PROGRAM P_Sortierer
VAR
END_VAR

(* 
Baustein: FC24 Sortierer
Zeitstempel Code: 25.06.2018 11:16:45
Interface: 27.09.2011 10:59:21
*)

F_Sortierer(); //OK

F_Vereinzelung(); //SV noch den block verwenden

F_Leerfahren(); //OK

END_PROGRAM

(* stored: Version 1.1.0.1, ProductVersion 3.1.4024.3
   POU P_Sortierer: Id {65b34c3b-6004-40b5-a999-e2ce64598a68}, SpecialFunc None *)
